FUNCTION_BLOCK FBOscillator
VAR_INPUT
	tPeriodRise	: TIME;
	tPeriodFall	: TIME;
END_VAR
VAR_OUTPUT
	byValue	 AT %Q*	: BYTE;
END_VAR
VAR
	tonRise	: TON;
	tonFall : TON;
	MAXVALUE	: UDINT := 255;
	iCycle  : INT;
END_VAR

tonRise(PT	:= tPeriodRise);
tonFall(PT	:= tPeriodFall);

CASE iCycle OF
	
0:
tonRise.IN	:= TRUE;
iCycle		:= 10;

10:
IF tonRise.Q THEN
	tonRise.IN	:= FALSE;
	tonFall.IN	:= TRUE;
	iCycle		:= 20;
END_IF

20:
IF tonFall.Q THEN
	tonFall.IN	:= FALSE;
	iCycle		:= 0;
END_IF

END_CASE

IF tonRise.IN THEN
	byValue	:= UDINT_TO_BYTE(MAXVALUE);
ELSE
	byValue	:= 3;
END_IF

END_FUNCTION_BLOCK

(* stored: Version 1.1.0.1, ProductVersion 3.1.4024.9
   POU FBOscillator: Id {ed8238c6-74da-4734-b807-ea1870f7ed7e}, SpecialFunc None *)
